(* PLC project  *)

PROGRAM P
  VAR  (* added by the conversion: wires and edge detectors of the diagram *)
    _GT3_ENO : BOOL;
    _GT3_OUT : BOOL;
    _MUL6_ENO : BOOL;
    _MUL6_OUT : ANY;
    _MOVE4_ENO : BOOL;
    _MOVE4_OUT : ANY;
  END_VAR

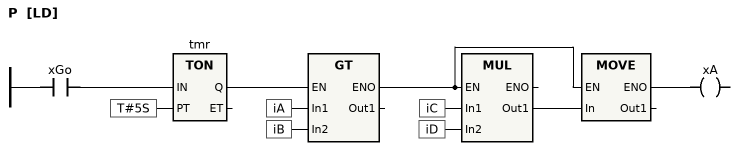
(* LD diagram, written out as Structured Text *)
tmr(IN := xGo, PT := T#5S);
_GT3_OUT := GT(EN := tmr.Q, IN1 := iA, IN2 := iB, ENO => _GT3_ENO);
_MUL6_OUT := MUL(EN := _GT3_ENO, IN1 := iC, IN2 := iD, ENO => _MUL6_ENO);
_MOVE4_OUT := MOVE(EN := _GT3_ENO, In := _MUL6_OUT, ENO => _MOVE4_ENO);
xA := _MOVE4_ENO;
END_PROGRAM
